TYPE ST_DeviceSingleChannelInput :
STRUCT
	stSafetyDescription : ST_SafetyDescription;
	Output AT %I* : BOOL;
END_STRUCT
END_TYPE

(* stored: Version 1.1.0.1, ProductVersion 3.1.4026.18
   DUT ST_DeviceSingleChannelInput: Id {72112c5f-9fd9-4db3-9116-86c6d930c50a} *)
